{attribute addProperty BoxType "EL6201-0000-0017"}
{attribute addProperty Id "Slave_30A_DI0BIT10.125233Slave_30A_DI1BIT10.125234Slave_30A_DI2BIT10.125235Slave_30A_DI3BIT10.125236Slave_30B_DI0BIT10.125237Slave_30B_DI1BIT10.125238Slave_30B_DI2BIT10.125239Slave_30B_DI3BIT10.125240"}
{attribute addProperty CRC "294374527"}
{attribute addProperty SizeInBites "8"}
{attribute addProperty SizeInBytes "1"}
TYPE Slave_30_Inputs_118BCC7F :
STRUCT
	{attribute addProperty Name "Slave_30A_DI0"}
	Slave_30A_DI0 : BIT;
	{attribute addProperty Name "Slave_30A_DI1"}
	Slave_30A_DI1 : BIT;
	{attribute addProperty Name "Slave_30A_DI2"}
	Slave_30A_DI2 : BIT;
	{attribute addProperty Name "Slave_30A_DI3"}
	Slave_30A_DI3 : BIT;
	{attribute addProperty Name "Slave_30B_DI0"}
	Slave_30B_DI0 : BIT;
	{attribute addProperty Name "Slave_30B_DI1"}
	Slave_30B_DI1 : BIT;
	{attribute addProperty Name "Slave_30B_DI2"}
	Slave_30B_DI2 : BIT;
	{attribute addProperty Name "Slave_30B_DI3"}
	Slave_30B_DI3 : BIT;
END_STRUCT
END_TYPE

(* stored: Version 1.2.0.0, ProductVersion 3.1.4024.9
   DUT Slave_30_Inputs_118BCC7F: Id {2115b452-c60a-488f-8144-72d4eef5544e} *)
